FUNCTION_BLOCK L2_StateTracker (* Basic Function Block Type *)
  (* Standard: 61499-2 *)
  (* Version 0.0, 2014-12-04, EQUEROL, UJI *)
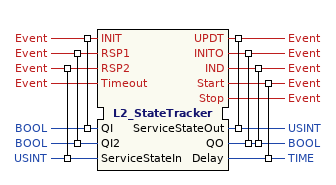
  EVENT_INPUT
    INIT WITH QI; (* Service Initialization Request *)
    RSP1 WITH QI2; (* Service response to initialization *)
    RSP2 WITH ServiceStateIn; (* Service state request response *)
    Timeout; (* Delay timeout *)
  END_EVENT
  EVENT_OUTPUT
    UPDT WITH ServiceStateOut; (* Update Machine state *)
    INITO WITH QO; (* Indicate Service to change state *)
    IND WITH QO; (* Request machine service state *)
    Start WITH Delay; (* Timeout start *)
    Stop; (* Timeout stop *)
  END_EVENT
  VAR_INPUT
    QI : BOOL; (* Input event qualifier *)
    QI2 : BOOL; (* Input event qualifier *)
    ServiceStateIn : USINT; (* Machine service state *)
  END_VAR
  VAR_OUTPUT
    ServiceStateOut : USINT; (* Machine service state *)
    QO : BOOL; (* Output event qualifier *)
    Delay : TIME; (* Timeout delay *)
  END_VAR
  VAR
    TOCounter : USINT := 0; (* Timeouts counter *)
    MaxTO : USINT := 10; (* Maximum number fo timeouts *)
    ServiceWorking : BOOL := FALSE; (* This flag indicates if the service is supposed to be running or not *)
  END_VAR
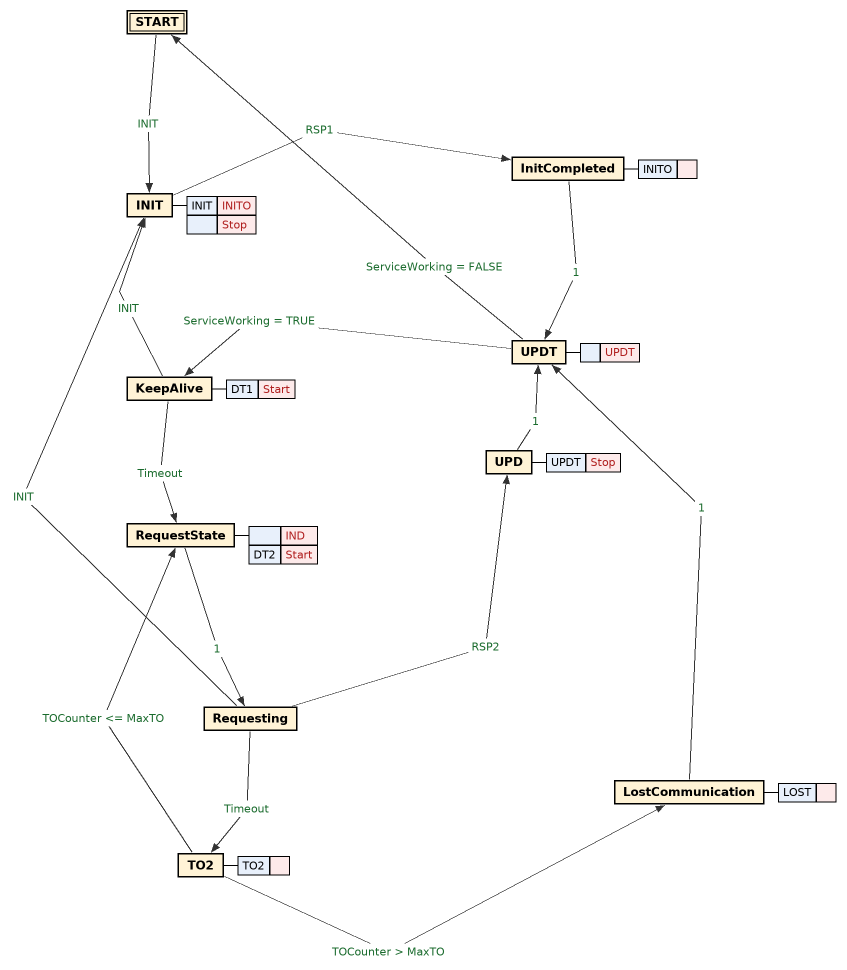
  EC_STATES
    START; (* Initial State *)
    INIT : INIT -> INITO, -> Stop; (* Initialization *)
    UPDT : -> UPDT; (* Normal execution *)
    InitCompleted : INITO;
    UPD : UPDT -> Stop;
    RequestState : -> IND, DT2 -> Start;
    KeepAlive : DT1 -> Start;
    Requesting;
    TO2 : TO2;
    LostCommunication : LOST;
  END_STATES
  EC_TRANSITIONS
    START TO INIT := INIT;
    InitCompleted TO UPDT := 1;
    UPD TO UPDT := 1;
    RequestState TO Requesting := 1;
    KeepAlive TO RequestState := Timeout;
    Requesting TO UPD := RSP2;
    UPDT TO KeepAlive := ServiceWorking = TRUE;
    INIT TO InitCompleted := RSP1;
    Requesting TO TO2 := Timeout;
    TO2 TO RequestState := TOCounter <= MaxTO;
    TO2 TO LostCommunication := TOCounter > MaxTO;
    LostCommunication TO UPDT := 1;
    UPDT TO START := ServiceWorking = FALSE;
    KeepAlive TO INIT := INIT;
    Requesting TO INIT := INIT;
  END_TRANSITIONS
  ALGORITHM INIT IN ST: (* Initialization algorithm *)
IF QI = TRUE THEN
	QO := TRUE;
ELSE
	QO := FALSE;
END_IF;
  END_ALGORITHM
  ALGORITHM UPDT IN ST: (* Update service state algo *)
ServiceStateOut := ServiceStateIn;
(*Reset timeouts counter*)
TOCounter := 0;
  END_ALGORITHM
  ALGORITHM INITO IN ST: (* Initialization completed algo *)
(*This algo is called once the machine initialization is completed*)
IF QI2 = TRUE THEN
	(*Initialization succed*)
	ServiceStateOut := 1;
	ServiceWorking := TRUE;
ELSE
	ServiceStateOut := 0;
	ServiceWorking := FALSE;
END_IF;
  END_ALGORITHM
  ALGORITHM DT1 IN ST: (* Keep alive algo *)
(*Periodic machine check*)
Delay := TIME#60000ms;
  END_ALGORITHM
  ALGORITHM DT2 IN ST: (* REQS algo *)
(*A Machine is expected to answer within a second to a request state event*)
Delay := TIME#1000ms;
  END_ALGORITHM
  ALGORITHM TO2 IN ST: (* Algorithm to control the number fo timeouts while requesting the service state *)
TOCounter := TOCounter + 1;
  END_ALGORITHM
  ALGORITHM LOST IN ST: (* lost communication algo *)
(*We lost the communication with the Machine service*)
ServiceStateOut :=  0;
  END_ALGORITHM
END_FUNCTION_BLOCK
